Fanuc KAREL source: ko00076.KL

-- PROVISIONAL review KL for V770-1; original PC SHA256 252470a4dad3e94aa0d9fefe42bf40b788f7c5f9c6b08c984542774d3d81f51b
-- Incomplete behavior may be omitted. Consult companion uncertainty JSON. Do not deploy.
PROGRAM KO00076
%NOLOCKGROUP
BEGIN
  -- UNRESOLVED_PC offsets 5-12; opcodes 9D,23
  -- UNRESOLVED_PC offsets 17-66; opcodes 27,22,1C,27,49,7E,AD,22,31,7E,4A
  -- UNRESOLVED_PC offsets 71-75; opcodes 7F
END KO00076
